Fanuc KAREL source: kb00050.KL

PROGRAM KB00050
%STACKSIZE=65535
%PRIORITY=65535
%NOLOCKGROUP
VAR
P1 : STRING[80]
P2 : STRING[80]
P3 : STRING[80]
P4 : STRING[80]
P5 : INTEGER
P6 : INTEGER
P7 : INTEGER
P8 : INTEGER
P9 : INTEGER
BEGIN
P1='A'
P2='A'
P3='A'
P4='A'
P5=1
P6=1
P7=1
P8=1
P9=1
CREATE_VAR(P1,P2,P3,P4,P5,P6,P7,P8,P9,1)
END KB00050
